{attribute 'strict'}
TYPE MoverCommandType_enum : (
        MOVETYPE_NONE     		:= 0,
        MOVETYPE_POSITION		:= 1,
        MOVETYPE_STATION 		:= 2,
        MOVETYPE_VELOCITY 		:= 3,
        MOVETYPE_SYNC_MOVER     := 4,
		MOVETYPE_SYNC_AXIS		:= 5,
		MOVETYPE_MULTISTATION	:= 6
    );
END_TYPE

(* stored: Version 1.1.0.1, ProductVersion 3.1.4024.12
   DUT MoverCommandType_enum: Id {cfb76be7-0d79-49cb-87ba-a046be8c33bb} *)
